{attribute 'linkalways'} 
{attribute 'no_explicit_call' := 'This FB is a CLASS and must be accessed using methods or properties'}
{attribute 'enable_dynamic_creation'}
FUNCTION_BLOCK FINAL EQ_USINT EXTENDS Node
VAR
	in1 : _USINT(0);
	in2 : _USINT(0);
	out : _BOOL(FALSE);
END_VAR

METHOD PUBLIC Clone : I_Node
VAR
	pNode : POINTER TO EQ_USINT;
END_VAR
pNode := __NEW(EQ_USINT);
Clone := pNode^;
END_METHOD

METHOD FB_init : BOOL
VAR_INPUT
	bInitRetains : BOOL; // if TRUE, the retain variables are initialized (warm start / cold start)
	bInCopyCode : BOOL;  // if TRUE, the instance afterwards gets moved into the copy code (online change)
END_VAR
AddInput('in1',THIS^.in1);
AddInput('in2',THIS^.in2);
AddOutput('out', THIS^.out);
END_METHOD

METHOD PROTECTED OnExecute
VAR
END_VAR
out.Value := in1.Value = in2.Value;
END_METHOD

END_FUNCTION_BLOCK

(* stored: Version 1.1.0.1, ProductVersion 3.1.4024.15
   POU EQ_USINT: Id {a08d852c-3801-470f-951a-00368d78ee7c}, SpecialFunc None
   Folder Constructor: Id {c59095b4-b609-4aa8-a5a3-35a8da87b1a0}
   Method Clone: Id {760077b1-1f4b-4ba1-aee4-5dca81b4f95d}
   Method FB_init: Id {b6912162-5d9a-4341-a6ab-72fe9c122ec0}
   Method OnExecute: Id {5f2f7177-937f-4d82-9a6b-1f65f8dcc1bb} *)
